(* PLC project CoDeSys External Library Template, WAGO e!COCKPIT e!COCKPIT, author 3S - Smart Software Solutions GmbH *)
(* stored: creationDateTime 2019-10-29T12:37:19.6052652, version 3.5.5.30, modificationDateTime 2019-10-29T12:36:39.3744516, organization 3S - Smart Software Solutions GmbH *)
(* Library project template with all possible element types, docu and a sample project structure *)

(* Nazwa bloku: Blok funkcyjny konwersji liczby decymalnej na binarną Autor: Jan Bartczak Wersja: v1.0.0 - 2018-06-22 *)
FUNCTION_BLOCK fbDecToBin
  VAR_INPUT
    wWordWejsciowy : WORD;
    intIloscBitow : INT;
  END_VAR
  VAR_OUTPUT
    arBity : ARRAY[0..16] OF BYTE;
  END_VAR
  VAR
    intWejsciowy : UINT;
    bBajtPojedynczy : BYTE;
    intWord : WORD;
    intI : INT;
  END_VAR

            intWejsciowy := WORD_TO_UINT(wWordWejsciowy);
intIloscBitow := intIloscBitow - 1;
FOR intI := 0 TO intIloscBitow BY 1 DO
	intWord := (intWejsciowy MOD 2);
	bBajtPojedynczy := UINT_TO_BYTE(intWord);
	arBity[intI] := bBajtPojedynczy;
	intWejsciowy := intWejsciowy/2;
END_FOR;

          
END_FUNCTION_BLOCK
